Fanuc KAREL source: CLOSE_TPE.kl

PROGRAM T
%NOLOCKGROUP
VAR
 v0 : INTEGER
 v1 : INTEGER
BEGIN
 CLOSE_TPE(v0, v1)
END T
